TYPE TupleStruct_4:
    STRUCT
        field0: DINT;
        field1: DINT;
        field2: DINT;
        field3: DINT;
        field4: DINT;
        field5: DINT;
        field6: DINT;
        field7: DINT;
        field8: DINT;
        field9: DINT;
        field10: DINT;
        field11: DINT;
        field12: DINT;
        field13: DINT;
        field14: DINT;
        field15: DINT;
        field16: DINT;
        field17: DINT;
        field18: DINT;
        field19: DINT;
        field20: DINT;
        field21: DINT;
        field22: DINT;
        field23: DINT;
        field24: DINT;
        field25: DINT;
        field26: DINT;
        field27: DINT;
        field28: DINT;
        field29: DINT;
        field30: DINT;
        field31: DINT;
        field32: DINT;
        field33: DINT;
        field34: DINT;
    END_STRUCT
END_TYPE

(* stored: ProductVersion 3.1.0.18, Version 1.1.0.1 *)
